// TIA Portal V20 export
TYPE "ConveyorStatus"
// stored: Access Published, Namespace Global
   STRUCT
      Blockage : Bool;
      xReserved_2 : Bool;
      xReserved_3 : Bool;
      xReserved_4 : Bool;
      xReserved_5 : Bool;
      xReserved_6 : Bool;
      xReserved_7 : Bool;
      xReserved_8 : Bool;
      ON : Bool;
      ReadytoRun : Bool;
      Occupied : Bool;
      Running : Bool;
      Fault : Bool;
      Estop : Bool;
      Manual : Bool;
      Stop : Bool;
   END_STRUCT;
END_TYPE
